FUNCTION_BLOCK logiBUS_ID (* Input service interface function block for double word input data *)
  (* Description: Copyright (c) 2017 fortiss GmbH, HR Agrartechnik GmbH This program and the accompanying materials are made available under the terms of the Eclipse Public License 2.0 which is available at https://www.eclipse.org/legal/epl-2.0/ SPDX-License-Identifier: EPL-2.0 this works for: BUTTON_PRESS_UP BUTTON_LONG_PRESS_HOLD BUTTON_LONG_PRESS_UP *)
  (* Version 1.0, 2017-03-20, Monika Wenger, fortiss GmbH, initial API and implementation and/or initial documentation *)
  PACKAGE logiBUS::io::DI;
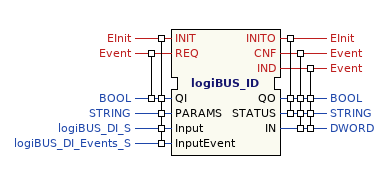
  EVENT_INPUT
    INIT : EInit WITH QI, PARAMS, Input, InputEvent; (* Service Initialization *)
    REQ WITH QI; (* Service Request *)
  END_EVENT
  EVENT_OUTPUT
    INITO : EInit WITH QO, STATUS; (* Initialization Confirm *)
    CNF WITH QO, STATUS, IN; (* Confirmation of Requested Service *)
    IND WITH QO, STATUS, IN; (* Indication from Resource *)
  END_EVENT
  VAR_INPUT
    QI : BOOL; (* Event Input Qualifier *)
    PARAMS : STRING; (* Service Parameters *)
    Input : logiBUS::io::DI::logiBUS_DI_S := logiBUS_DI::Invalid; (* Identify the Input Input_I1..I8 *)
    InputEvent : logiBUS::io::DI::logiBUS_DI_Events_S := logiBUS_DI_Events::Invalid; (* Identify the Event (currently only REPEAT supported) *)
  END_VAR
  VAR_OUTPUT
    QO : BOOL; (* Event Output Qualifier *)
    STATUS : STRING; (* Service Status *)
    IN : DWORD; (* Input data from resource *)
  END_VAR
END_FUNCTION_BLOCK
